TYPE ST_IndexedPositionControls :
	STRUCT
		// Operating modes
		OperationMode		: BOOL := FALSE; // TRUE = Automatic, FALSE = Manual
		isDefined 			: BOOL := FALSE; // Change to true if this position exists
		State				: E_IndexedPositionStates := E_IndexedPositionStates.Starved;
		Request				: E_IndexedPositionTransitionRequest := E_IndexedPositionTransitionRequest.NoRequest;
		
		// Sensing
		ArrivalDetection	: BOOL;
		AreaMonitoring		: BOOL;

		// Internal Directional Controls for Linking
		Front				: ST_DirectionalControls;
		Rear				: ST_DirectionalControls;
		Left				: ST_DirectionalControls;
		Right				: ST_DirectionalControls;
		
	END_STRUCT
END_TYPE

(* stored: Version 1.1.0.1, ProductVersion 3.1.4024.12
   DUT ST_IndexedPositionControls: Id {d7bb33da-6062-4bf2-a354-bc140dc5ad12} *)
